ABB RobotStudio station: Tp2_20201214-032332.rsstn

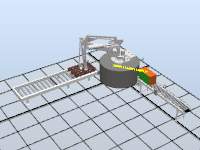
Station Tp2 (saved by RobotStudio 20.2.9116.0)
Controller Controlador1
  mechanical unit ROB_1: IRB660_180_315__01_2, 6 joints, base frame (0, 0, 1000) mm
Layout (positions relative to the parent item):
  - transporteCajas [part, from Equipment\Conveyor Guide 400.rslib] at (0, 1500, 0) mm, rotated rx 0 ry 0 rz 90 deg
  - Euro Pallet [graphiccomponentgroup, from Equipment\Euro Pallet.rslib] at (1000, -1425, 435) mm
    - Body 1 [part, from Equipment\Euro Pallet.rslib]
  - transportePallets [part, from Equipment\Conveyor 950 4000 h2.rslib] at (1000, -1500, 0) mm
  - caja [part] at (-200, 1500, 770) mm
  - IRB660_180_315__01_2 [mechanism, from Robots\IRB660_180_315__01.rslib] at (0, 0, 1000) mm; joint values [1.7033, -0.0683, 0.6907, 1.7033] (rad or m)
  - ventosa_tool [mechanism] at (1662.34, -987.3, 320.65) mm, rotated rx 180 ry 0 rz 180 deg
      TCP ventosa_tool at (0, 0, 200) mm
      links: ventosa
  - pedestal [part]
Attachment: Euro Pallet is attached to transportePallets
Attachment: ventosa_tool is attached to IRB660_180_315__01_2 / Link6
Attachment: pistaCajas is attached to transporteCajas
Attachment: pistaPallets is attached to transportePallets
EventTableEntry 2069: Group=, Trigger=do_pick 2070, Actions=[EventTableActionAttach 2071], Comment=, ActivationMode=2, Cyclic=false
EventTableTriggerIO 2070: IOValue=[1], IRC5Controller=? -1, Operator=0, SignalSource=Controlador1 1586
EventTableActionAttach 2071: AttachmentParent=ventosa_tool 1580, AttachmentChild=caja 1044, MountObject=false, Offset=[X=1, Y=0, Z=0, W=0, X=0, Y=1, Z=0, W=0, X=0, Y=0, Z=1, W=0, X=0, Y=0, Z=0, W=1], FlangeIndext=0, FindNearest=false
EventTableEntry 2072: Group=, Trigger=do_pick 2073, Actions=[EventTableActionDetach 2074], Comment=, ActivationMode=2, Cyclic=false
EventTableTriggerIO 2073: IOValue=[0], IRC5Controller=? -1, Operator=0, SignalSource=Controlador1 1586
EventTableActionDetach 2074: AttachmentParent=ventosa_tool 1580, AttachmentChild=caja 1044
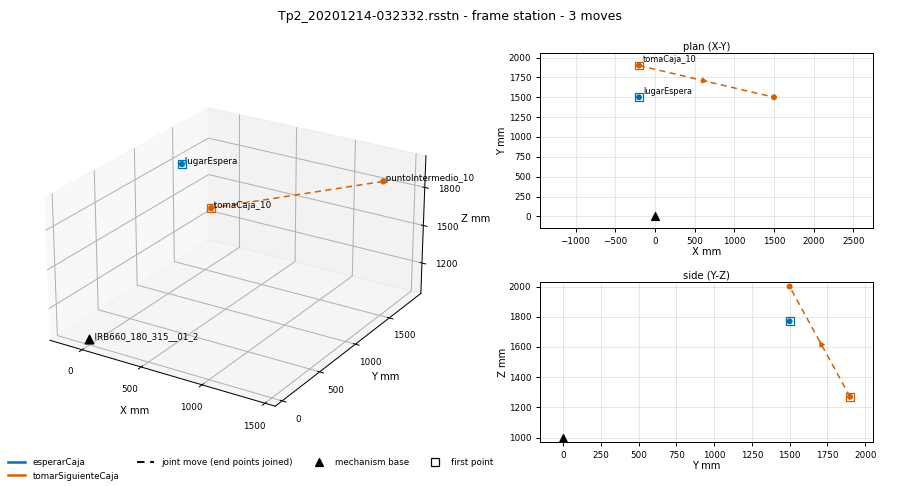
[picture p0: tool path of Tp2_20201214-032332.rsstn in frame station, 3 of 3 moves have a stored position in this frame; points joined in program order, loops and branches not executed]
Targets, tools, work objects and paths stored in the station, written as RAPID:
! task T_ROB1
MODULE Module1
  PERS tooldata ventosa_tool:=[TRUE,[[0,0,200],[1,0,0,0]],[1,[0,0,1],[1,0,0,0],0,0,0]];
  PERS wobjdata pistaCajas:=[FALSE,TRUE,"",[[-200,1500,770],[0,0,1,0]],[[0,0,0],[1,0,0,0]]];
  PERS wobjdata pistaPallets:=[FALSE,TRUE,"",[[1000,-1425,579],[0,0,1,0]],[[0,0,0],[1,0,0,0]]];
  CONST robtarget lugarEspera:=[[0,0,-1000],[1,0,0,0],[0,0,0,0],[9E+09,9E+09,9E+09,9E+09,9E+09,9E+09]];
  CONST robtarget tomaCaja_10:=[[0,400,-500],[1,0,0,0],[0,0,0,0],[9E+09,9E+09,9E+09,9E+09,9E+09,9E+09]];
  CONST robtarget superficiePallet_10:=[[0,0,0],[1,0,0,0],[0,0,0,0],[9E+09,9E+09,9E+09,9E+09,9E+09,9E+09]];
  CONST robtarget puntoIntermedio_10:=[[1500,1500,2000],[0,0,1,0],[0,0,0,0],[9E+09,9E+09,9E+09,9E+09,9E+09,9E+09]];
  PROC main()
    esperarCaja;
    tomarSiguienteCaja;
    esperarCaja;
  ENDPROC
  PROC esperarCaja()
    MoveJ lugarEspera,v1000,fine,ventosa_tool\WObj:=pistaCajas;
  ENDPROC
  PROC tomarSiguienteCaja()
    MoveJ tomaCaja_10,v1000,fine,ventosa_tool\WObj:=pistaCajas;
    SetDO do_pick,1;
    MoveJ puntoIntermedio_10,v1000,z100,ventosa_tool\WObj:=wobj0;
  ENDPROC
ENDMODULE

